// TIA Portal V17 export
VAR_GLOBAL   // PLC tag table "Default tag table"
   StartCmd AT %I0.0 : Bool;
END_VAR
